FUNCTION_BLOCK Handling_Positions EXTENDS TcoDrivesBeckhoff.TcoSingleAxisPositionsRootContainer

VAR
	{attribute addProperty Name "<#Pick Position#>"}
	PickPosition:TcoDrivesBeckhoff.TcoSIngleAxisMoveParam;
	{attribute addProperty Name "<#Place  Position#>"}
	PlacePosition:TcoDrivesBeckhoff.TcoSingleAxisMoveParam;
END_VAR

END_FUNCTION_BLOCK

(* stored: Version 1.1.0.1
   POU Handling_Positions: Id {e471d124-0d09-4412-a76e-60ce34f54752}, SpecialFunc None *)
